INTERFACE I_Interface

END_INTERFACE

(* stored: Version 1.1.0.1, ProductVersion 3.1.4024.3
   Itf I_Interface: Id {b6907b15-f762-4e07-b3e0-89eb3e4cddea} *)
